{attribute 'qualified_only'}
VAR_GLOBAL
	
	//all slaves
	EtherCATslaveDiag: ARRAY[1..maxNumEtherCATSlaves] OF typeEtherCATIndicator;

	//assign to mapped IO for DPstate
	RawDPStateDiag: ARRAY[1..maxNumEtherCATSlaves] OF USINT;

END_VAR



//UINT
//0x___1 = Slave in 'INIT' state
//0x___2 = Slave in 'PREOP' state
//0x___3 = Slave in 'BOOT' state
//0x___4 = Slave in 'SAFEOP' state
//0x___8 = Slave in 'OP' state
//0x001_ = Slave signals error
//0x002_ = Invalid vendorId, productCode... read
//0x004_ = Initialization error occurred
//0x008_ = Slave disabled
//0x010_ = Slave not present
//0x020_ = Slave signals link error
//0x040_ = Slave signals missing link
//0x080_ = Slave signals unexpected link
//0x100_ = Communication port A
//0x200_ = Communication port B
//0x400_ = Communication port C
//0x800_ = Communication port D



VAR_GLOBAL CONSTANT
	maxNumEtherCATSlaves: UINT := 65535;
END_VAR

(* stored: Version 1.1.0.1, ProductVersion 3.1.4024.12
   GVL etherCATdiag: Id {3f381e22-eb2f-465b-8c21-a28935184f16} *)
